FUNCTION_BLOCK DataPanel_STATUS_SAE_J1939 (* Status Output of 1 DataPanel Node *)
  (* Standard: SAE J1939; Description: Copyright (c) 2018, 2023 Jose Cabral, HR Agrartechnik GmbH This program and the accompanying materials are made available under the terms of the Eclipse Public License 2.0 which is available at https://www.eclipse.org/legal/epl-2.0/ SPDX-License-Identifier: EPL-2.0 *)
  (* Version 1.0, 2018-12-05, Jose Cabral *)
  (* Version 1.1, 2022-08-04, Franz Höpfinger, HR Agrartechnik GmbH *)
  (* Version 1.2, 2023-01-05, Franz Höpfinger, HR Agrartechnik GmbH *)
  PACKAGE DataPanel::Status;
  IMPORT DataPanel::io::MI::const::MI;
  IMPORT eclipse4diac::core::TypeHash;
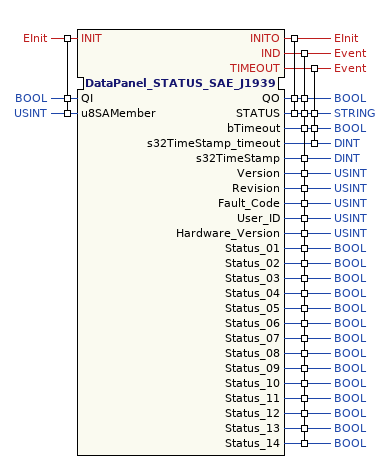
  EVENT_INPUT
    INIT : EInit WITH QI, u8SAMember; (* Service Initialization *)
  END_EVENT
  EVENT_OUTPUT
    INITO : EInit WITH QO, STATUS; (* Initialization Confirm *)
    IND WITH QO, s32TimeStamp, STATUS, bTimeout, Version, Revision, Fault_Code, User_ID, Hardware_Version, Status_01, Status_02, Status_03, Status_04, Status_05, Status_06, Status_07, Status_08, Status_09, Status_10, Status_11, Status_12, Status_13, Status_14; (* Indication from Resource *)
    TIMEOUT WITH s32TimeStamp_timeout, STATUS, bTimeout;
  END_EVENT
  VAR_INPUT
    QI : BOOL; (* Event Input Qualifier *)
    u8SAMember : USINT := MI::MI_00; (* Node SA 224..239 *)
  END_VAR
  VAR_OUTPUT
    QO : BOOL; (* Event Output Qualifier *)
    STATUS : STRING; (* Service Status *)
    bTimeout : BOOL := FALSE; (* Timeout occured TRUE = Timeout, FALSE = no Timeout *)
    s32TimeStamp_timeout : DINT;
    s32TimeStamp : DINT;
    Version : USINT;
    Revision : USINT;
    Fault_Code : USINT;
    User_ID : USINT;
    Hardware_Version : USINT;
    Status_01 : BOOL;
    Status_02 : BOOL;
    Status_03 : BOOL;
    Status_04 : BOOL;
    Status_05 : BOOL;
    Status_06 : BOOL;
    Status_07 : BOOL;
    Status_08 : BOOL;
    Status_09 : BOOL;
    Status_10 : BOOL;
    Status_11 : BOOL;
    Status_12 : BOOL;
    Status_13 : BOOL;
    Status_14 : BOOL;
  END_VAR
END_FUNCTION_BLOCK
